// SIMATIC S7-200 SMART project (STEP 7-Micro/WIN SMART), CPU SR40

SYMBOL_TABLE 系统符号
Always_On        SM0.0    // 始终接通
First_Scan_On    SM0.1    // 仅在第一个扫描周期时接通
IO_Err           SM5.0    // 存在任何 I/O 错误时置位为 1
END_SYMBOL_TABLE

ORGANIZATION_BLOCK MAIN:OB1
TITLE=程序注释
BEGIN
Network 1
// 程序段注释
LD     First_Scan_On:SM0.1
ATCH   INT_0:INT0, 0
ATCH   INT_1:INT1, 3
ENI
Network 2
LD     IO_Err:SM5.0
DTCH   0
DTCH   3
END_ORGANIZATION_BLOCK

INTERRUPT_BLOCK INT_0:INT0
TITLE=中断例程注释
BEGIN
Network 1
// 程序段注释
LD     Always_On:SM0.0
SI     Q0.0, 1
TODR   VB10
END_INTERRUPT_BLOCK

INTERRUPT_BLOCK INT_1:INT1
TITLE=中断例程注释
BEGIN
Network 1
// 程序段注释
LD     Always_On:SM0.0
RI     Q0.0, 1
TODR   VB18
END_INTERRUPT_BLOCK
